FUNCTION_BLOCK FB_Button
VAR
	sButtonName : STRING;
	bExecute : BOOL;
	ExecuteCounter : UDINT;
	refCommand : REFERENCE TO E_Command;
	InputCommand : E_Command;
	
	bInit : BOOL;
END_VAR

IF bExecute THEN
	ExecuteCounter := ExecuteCounter + _TaskInfo[1].CycleTime/10000;
	IF ExecuteCounter >= 1000 THEN
		refCommand := InputCommand;
		bExecute := FALSE;
	END_IF
ELSE
	ExecuteCounter := 0;
END_IF

METHOD Initalize
VAR_IN_OUT
	refCommand : E_Command;
END_VAR
VAR_INPUT
	ButtonName : E_Command;
END_VAR
sButtonName := TO_STRING(ButtonName);
THIS^.InputCommand := ButtonName;
THIS^.refCommand REF= refCommand;
bInit := TRUE;
END_METHOD

END_FUNCTION_BLOCK

(* stored: Version 1.1.0.1, ProductVersion 3.1.4024.12
   POU FB_Button: Id {39098658-c1cc-443a-8bd8-27357fe3de3f}, SpecialFunc None
   Method Initalize: Id {cfe61e61-c2a3-40f8-9404-95b0b7ed5754} *)
